Yaskawa INFORM job: FRONT_SEARCH_-90ST-2_4740.JBI

/JOB
//NAME FRONT_SEARCH_-90ST-2_4740
///FOLDERNAME 02-SKRZYNIE_JOBS
//POS
///NPOS 61,61,0,9,0,0
///TOOL 0
///POSTYPE PULSE
///PULSE
C00000=-14334,-10708,45002,-95286,-40321,-4878
C00001=-1,-11355,44471,-89821,-32839,-4429
C00002=51470,-3981,47579,-58794,-5299,-8788
C00003=55570,1468,42458,-7386,-9208,-33373
C00004=67803,1091,42035,59104,-16935,-61314
C00005=66620,9721,53664,53490,-17138,-58745
C00006=65132,11491,55975,50657,-16585,-57605
C00007=66620,9721,53664,53490,-17138,-58745
C00008=67271,11853,56546,53440,-17675,-58611
C00009=54816,3282,46487,30906,-12207,-49746
C00010=54816,6101,53312,25756,-14460,-47262
C00011=59008,-4535,34194,48609,-11906,-57578
C00012=69764,-14576,19632,71385,-22274,-9844
C00013=70020,-17345,11989,86916,-25690,33597
C00014=67336,-3926,30729,80145,-24196,36739
C00015=66500,-3667,31093,79640,-23688,36879
C00016=65119,-2468,32336,79080,-22832,36966
C00017=65297,-2627,32170,79156,-22942,36953
C00018=65297,-1325,35513,76192,-23171,38468
C00019=66289,-3938,30110,80584,-23496,36363
C00020=51768,-18636,16430,81328,-29399,37370
C00021=49437,-15984,19531,80095,-27994,37663
C00022=48263,-14852,20450,79978,-27248,37540
C00023=48412,-15000,20329,79992,-27342,37556
C00024=48412,-13851,23216,77920,-27509,38655
C00025=49631,-16164,19389,80113,-28114,37684
C00026=53676,-11243,23565,89149,-42613,36486
C00027=52851,-10439,24283,89045,-42108,36402
C00028=53146,-10730,24020,89082,-42288,36431
C00029=53146,-9547,27031,87832,-42262,37235
C00030=54384,-12125,22415,89467,-43055,36413
C00031=34191,-19915,16180,80853,-30719,37960
C00032=33662,-19058,17079,80673,-30395,37970
C00033=32807,-17866,17978,80777,-29844,37774
C00034=32930,-18043,17844,80762,-29923,37803
C00035=32930,-16777,20995,78746,-30087,38900
C00036=34005,-19810,16015,81091,-30585,37800
C00037=3145,-18728,16815,77374,-25054,38329
C00038=817,-17844,18158,75547,-23707,38913
C00039=796,-16604,19121,76122,-23639,38615
C00040=799,-16751,19005,76056,-23647,38649
C00041=799,-15711,21605,73897,-23867,39758
C00042=817,-18167,17401,76150,-23651,38603
C00043=-15498,-15616,13350,94001,-19148,32414
C00044=-15498,-15493,13676,93634,-19133,32596
C00045=-15205,-14385,14604,94183,-19340,32357
C00046=-15381,-15057,14039,93855,-19215,32498
C00047=-15381,-14074,16642,90939,-19118,33949
C00048=-15381,-15057,14039,93855,-19215,32498
C00049=-33931,-11015,21239,70432,-10097,42333
C00050=-33931,-10804,21788,69296,-10165,42874
C00051=-32905,-8952,23489,71704,-10712,41858
C00052=-32538,-11240,17958,92730,-11256,31526
C00053=-32538,-9785,21821,85083,-11210,35185
C00054=-32538,-11240,17958,92730,-11256,31526
C00055=-28620,-8047,30448,54655,-21030,45617
C00056=-30781,-7430,31038,52169,-19923,46526
C00057=-14004,-13983,22221,69587,-28542,40219
C00058=7437,-33768,-14250,91365,-41045,30812
C00059=0,-35574,42087,-36666,-9339,-1809
C00060=0,-52278,40443,0,6873,-1
BC00000=745522
BC00001=813007
BC00002=857017
BC00003=908607
BC00004=908607
BC00005=908607
BC00006=908607
BC00007=908607
BC00008=908607
BC00009=908608
BC00010=908608
BC00011=908608
BC00012=908608
BC00013=908608
BC00014=908608
BC00015=908608
BC00016=908608
BC00017=908608
BC00018=908608
BC00019=908960
BC00020=908960
BC00021=908960
BC00022=908960
BC00023=908960
BC00024=908960
BC00025=908960
BC00026=908960
BC00027=908960
BC00028=908960
BC00029=908960
BC00030=908960
BC00031=908960
BC00032=908960
BC00033=908960
BC00034=908960
BC00035=908960
BC00036=908960
BC00037=908960
BC00038=908960
BC00039=908960
BC00040=908960
BC00041=908960
BC00042=908960
BC00043=908960
BC00044=908960
BC00045=908960
BC00046=908960
BC00047=908960
BC00048=908960
BC00049=908960
BC00050=908960
BC00051=908960
BC00052=908960
BC00053=908960
BC00054=908960
BC00055=908960
BC00056=908960
BC00057=908960
BC00058=908960
BC00059=735553
BC00060=728676
///POSTYPE BASE
///RECTAN
///RCONF 1,0,0,0,0,0,0,0,0,0,0,0,0,0,0,0,0,0,0,0,0,0,0,0
P00006=0.000,0.000,0.000,0.0000,0.0000,0.0000
P00500=2.332,-5.281,-1.258,0.0000,0.0000,0.0000
///RCONF 0,0,0,0,0,0,0,0,0,0,0,0,0,0,0,0,0,0,0,0,0,0,0,0
P00501=-2.026,0.009,3.534,0.0000,0.0000,0.0000
///RCONF 1,0,0,0,0,0,0,0,0,0,0,0,0,0,0,0,0,0,0,0,0,0,0,0
P00502=-2.023,0.001,1.732,0.0000,0.0000,0.0000
P00503=0.138,-0.044,1.539,0.0000,0.0000,0.0000
P00504=-0.309,-0.010,1.636,0.0000,0.0000,0.0000
P00505=0.999,-9.916,8.214,0.0000,0.0000,0.0000
P00506=-2.492,-6.886,2.340,0.0000,0.0000,0.0000
P00510=-2.092,-0.040,5.096,0.0000,0.0000,0.0000
//INST
///DATE 2025/01/31 10:04
///ATTR SC,RW
///GROUP1 RB1,BS1
NOP
MOVJ C00000 BC00000 VJ=30.00
MOVJ C00001 BC00001 VJ=50.00
MOVJ C00002 BC00002 VJ=50.00
MOVJ C00003 BC00003 VJ=30.00
'::::::::::::::::::::::::::::::::
'W21 P
'::::::::::::::::::::::::::::::::
MOVL C00004 BC00004 V=333.3
MOVL C00005 BC00005 V=166.7 PL=0
REFP 3 C00006 BC00006
CALL JOB:SEARCH-R1
SET P0500 P0006
SFTON P0500
MOVL C00007 BC00007 V=166.7 PL=0
REFP 3 C00008 BC00008
CALL JOB:SEARCH-R1
SET P0500 P0006
SFTON P0500
MOVL C00009 BC00009 V=166.7 PL=0
REFP 3 C00010 BC00010
CALL JOB:SEARCH-R1
SET P0500 P0006
SFTOF
MOVL C00011 BC00011 V=166.7
'::::::::::::::::::::::::::::::::
'W21 L
'::::::::::::::::::::::::::::::::
MOVJ C00012 BC00012 VJ=50.00
MOVJ C00013 BC00013 VJ=70.00
MOVL C00014 BC00014 V=250.0
MOVL C00015 BC00015 V=166.7 PL=0
REFP 3 C00016 BC00016
CALL JOB:SEARCH-R1
SET P0501 P0006
SFTON P0501
MOVL C00017 BC00017 V=166.7 PL=0
REFP 3 C00018 BC00018
CALL JOB:SEARCH-R1
SET P0501 P0006
SFTON P0501
MOVL C00019 BC00019 V=166.7 PL=0
SFTOF
'::::::::::::::::::::::::::::::::
'W20 P
'::::::::::::::::::::::::::::::::
MOVL C00020 BC00020 V=333.3
MOVL C00021 BC00021 V=166.7 PL=0
REFP 3 C00022 BC00022
CALL JOB:SEARCH-R1
SET P0502 P0006
SFTON P0502
MOVL C00023 BC00023 V=166.7 PL=0
REFP 3 C00024 BC00024
CALL JOB:SEARCH-R1
SET P0502 P0006
SFTON P0502
MOVL C00025 BC00025 V=166.7 PL=0
SFTOF
MOVL C00026 BC00026 V=166.7 PL=0
REFP 3 C00027 BC00027
CALL JOB:SEARCH-R1
SET P0510 P0006
SFTON P0510
MOVL C00028 BC00028 V=66.7 PL=0
REFP 3 C00029 BC00029
CALL JOB:SEARCH-R1
SET P0510 P0006
SFTON P0510
MOVL C00030 BC00030 V=66.7 PL=0
SFTOF
'::::::::::::::::::::::::::::::::
'W20 L
'::::::::::::::::::::::::::::::::
MOVL C00031 BC00031 V=250.0
MOVL C00032 BC00032 V=166.7 PL=0
REFP 3 C00033 BC00033
CALL JOB:SEARCH-R1
SET P0503 P0006
SFTON P0503
MOVL C00034 BC00034 V=66.7 PL=0
REFP 3 C00035 BC00035
CALL JOB:SEARCH-R1
SET P0503 P0006
SFTON P0503
MOVL C00036 BC00036 V=166.7 PL=0
SFTOF
'::::::::::::::::::::::::::::::::
'W22 P
'::::::::::::::::::::::::::::::::
MOVL C00037 BC00037 V=333.3
MOVL C00038 BC00038 V=166.7 PL=0
REFP 3 C00039 BC00039
CALL JOB:SEARCH-R1
SET P0504 P0006
SFTON P0504
MOVL C00040 BC00040 V=66.7 PL=0
REFP 3 C00041 BC00041
CALL JOB:SEARCH-R1
SET P0504 P0006
SFTON P0504
MOVL C00042 BC00042 V=166.7 PL=0
SFTOF
'::::::::::::::::::::::::::::::::
'W22 L
'::::::::::::::::::::::::::::::::
MOVL C00043 BC00043 V=333.3
MOVL C00044 BC00044 V=166.7 PL=0
REFP 3 C00045 BC00045
CALL JOB:SEARCH-R1
SET P0505 P0006
SFTON P0505
MOVL C00046 BC00046 V=166.7 PL=0
REFP 3 C00047 BC00047
CALL JOB:SEARCH-R1
SET P0505 P0006
SFTON P0505
MOVL C00048 BC00048 V=166.7 PL=0
MOVL C00049 BC00049 V=333.3
MOVL C00050 BC00050 V=166.7
REFP 3 C00051 BC00051
CALL JOB:SEARCH-R1
SET P0506 P0006
SFTON P0506
MOVL C00052 BC00052 V=166.7
REFP 3 C00053 BC00053
CALL JOB:SEARCH-R1
SET P0505 P0006
SFTON P0506
MOVL C00054 BC00054 V=166.7
MOVL C00055 BC00055 V=166.7
REFP 3 C00056 BC00056
CALL JOB:SEARCH-R1
SET P0506 P0006
MOVL C00057 BC00057 V=333.3
MOVJ C00058 BC00058 VJ=50.00
SFTOF
MOVJ C00059 BC00059 VJ=80.00
MOVJ C00060 BC00060 VJ=80.00
END
